TYPE ST_Components_HMI_Command :
STRUCT
END_STRUCT
END_TYPE

(* stored: Version 1.1.0.1
   DUT ST_Components_HMI_Command: Id {b740f173-c501-09c3-1a6f-62d4925c2fd3} *)
